(* Visualisation Lamp_status
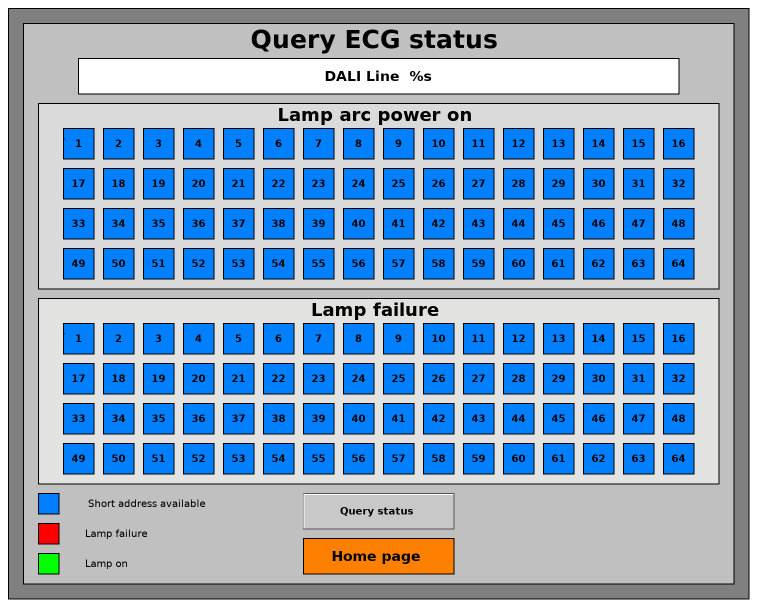
rectangle at (45,15)-(756,576): text "Query ECG status"
rounded rectangle at (325,530)-(476,566): text "Home page"; opens PLC_VISU; tooltip Back to home page
rounded rectangle at (100,50)-(701,86): text "DALI Line  %s"; shows DALI_Config.bDali_Linie; tooltip You can change the DALI Line only on the home page.
rectangle at (60,95)-(741,281): text "Lamp arc power on"
rectangle at (85,120)-(116,151): text "1"; alarm colour if DALI_Config.Kurzadr[1]
rectangle at (85,120)-(116,151): text "1"; invisible if not DALI_Config.Kurzadr[1]; alarm colour if DALI_Config.LampeEin[1]
rectangle at (125,120)-(156,151): text "2"; alarm colour if DALI_Config.Kurzadr[2]
rectangle at (125,120)-(156,151): text "2"; invisible if not DALI_Config.Kurzadr[2]; alarm colour if DALI_Config.LampeEin[2]
rectangle at (165,120)-(196,151): text "3"; alarm colour if DALI_Config.Kurzadr[3]
rectangle at (165,120)-(196,151): text "3"; invisible if not DALI_Config.Kurzadr[3]; alarm colour if DALI_Config.LampeEin[3]
rectangle at (205,120)-(236,151): text "4"; alarm colour if DALI_Config.Kurzadr[4]
rectangle at (205,120)-(236,151): text "4"; invisible if not DALI_Config.Kurzadr[4]; alarm colour if DALI_Config.LampeEin[4]
rectangle at (245,120)-(276,151): text "5"; alarm colour if DALI_Config.Kurzadr[5]
rectangle at (245,120)-(276,151): text "5"; invisible if not DALI_Config.Kurzadr[5]; alarm colour if DALI_Config.LampeEin[5]
rectangle at (285,120)-(316,151): text "6"; alarm colour if DALI_Config.Kurzadr[6]
rectangle at (285,120)-(316,151): text "6"; invisible if not DALI_Config.Kurzadr[6]; alarm colour if DALI_Config.LampeEin[6]
rectangle at (325,120)-(356,151): text "7"; alarm colour if DALI_Config.Kurzadr[7]
rectangle at (325,120)-(356,151): text "7"; invisible if not DALI_Config.Kurzadr[7]; alarm colour if DALI_Config.LampeEin[7]
rectangle at (365,120)-(396,151): text "8"; alarm colour if DALI_Config.Kurzadr[8]
rectangle at (365,120)-(396,151): text "8"; invisible if not DALI_Config.Kurzadr[8]; alarm colour if DALI_Config.LampeEin[8]
rectangle at (405,120)-(436,151): text "9"; alarm colour if DALI_Config.Kurzadr[9]
rectangle at (405,120)-(436,151): text "9"; invisible if not DALI_Config.Kurzadr[9]; alarm colour if DALI_Config.LampeEin[9]
rectangle at (445,120)-(476,151): text "10"; alarm colour if DALI_Config.Kurzadr[10]
rectangle at (445,120)-(476,151): text "10"; invisible if not DALI_Config.Kurzadr[10]; alarm colour if DALI_Config.LampeEin[10]
rectangle at (485,120)-(516,151): text "11"; alarm colour if DALI_Config.Kurzadr[11]
rectangle at (485,120)-(516,151): text "11"; invisible if not DALI_Config.Kurzadr[11]; alarm colour if DALI_Config.LampeEin[11]
rectangle at (525,120)-(556,151): text "12"; alarm colour if DALI_Config.Kurzadr[12]
rectangle at (525,120)-(556,151): text "12"; invisible if not DALI_Config.Kurzadr[12]; alarm colour if DALI_Config.LampeEin[12]
rectangle at (565,120)-(596,151): text "13"; alarm colour if DALI_Config.Kurzadr[13]
rectangle at (565,120)-(596,151): text "13"; invisible if not DALI_Config.Kurzadr[13]; alarm colour if DALI_Config.LampeEin[13]
rectangle at (605,120)-(636,151): text "14"; alarm colour if DALI_Config.Kurzadr[14]
rectangle at (605,120)-(636,151): text "14"; invisible if not DALI_Config.Kurzadr[14]; alarm colour if DALI_Config.LampeEin[14]
rectangle at (645,120)-(676,151): text "15"; alarm colour if DALI_Config.Kurzadr[15]
rectangle at (645,120)-(676,151): text "15"; invisible if not DALI_Config.Kurzadr[15]; alarm colour if DALI_Config.LampeEin[15]
rectangle at (685,120)-(716,151): text "16"; alarm colour if DALI_Config.Kurzadr[16]
rectangle at (685,120)-(716,151): text "16"; invisible if not DALI_Config.Kurzadr[16]; alarm colour if DALI_Config.LampeEin[16]
rectangle at (85,160)-(116,191): text "17"; alarm colour if DALI_Config.Kurzadr[17]
rectangle at (85,160)-(116,191): text "17"; invisible if not DALI_Config.Kurzadr[17]; alarm colour if DALI_Config.LampeEin[17]
rectangle at (165,160)-(196,191): text "19"; alarm colour if DALI_Config.Kurzadr[19]
rectangle at (165,160)-(196,191): text "19"; invisible if not DALI_Config.Kurzadr[19]; alarm colour if DALI_Config.LampeEin[19]
rectangle at (125,160)-(156,191): text "18"; alarm colour if DALI_Config.Kurzadr[18]
rectangle at (125,160)-(156,191): text "18"; invisible if not DALI_Config.Kurzadr[18]; alarm colour if DALI_Config.LampeEin[18]
rectangle at (205,160)-(236,191): text "20"; alarm colour if DALI_Config.Kurzadr[20]
rectangle at (205,160)-(236,191): text "20"; invisible if not DALI_Config.Kurzadr[20]; alarm colour if DALI_Config.LampeEin[20]
rectangle at (245,160)-(276,191): text "21"; alarm colour if DALI_Config.Kurzadr[21]
rectangle at (245,160)-(276,191): text "21"; invisible if not DALI_Config.Kurzadr[21]; alarm colour if DALI_Config.LampeEin[21]
rectangle at (285,160)-(316,191): text "22"; alarm colour if DALI_Config.Kurzadr[22]
rectangle at (285,160)-(316,191): text "22"; invisible if not DALI_Config.Kurzadr[22]; alarm colour if DALI_Config.LampeEin[22]
rectangle at (325,160)-(356,191): text "23"; alarm colour if DALI_Config.Kurzadr[23]
rectangle at (325,160)-(356,191): text "23"; invisible if not DALI_Config.Kurzadr[23]; alarm colour if DALI_Config.LampeEin[23]
rectangle at (365,160)-(396,191): text "24"; alarm colour if DALI_Config.Kurzadr[24]
rectangle at (365,160)-(396,191): text "24"; invisible if not DALI_Config.Kurzadr[24]; alarm colour if DALI_Config.LampeEin[24]
rectangle at (405,160)-(436,191): text "25"; alarm colour if DALI_Config.Kurzadr[25]
rectangle at (405,160)-(436,191): text "25"; invisible if not DALI_Config.Kurzadr[25]; alarm colour if DALI_Config.LampeEin[25]
rectangle at (565,160)-(596,191): text "29"; alarm colour if DALI_Config.Kurzadr[29]
rectangle at (565,160)-(596,191): text "29"; invisible if not DALI_Config.Kurzadr[29]; alarm colour if DALI_Config.LampeEin[29]
rectangle at (525,160)-(556,191): text "28"; alarm colour if DALI_Config.Kurzadr[28]
rectangle at (525,160)-(556,191): text "28"; invisible if not DALI_Config.Kurzadr[28]; alarm colour if DALI_Config.LampeEin[28]
rectangle at (485,160)-(516,191): text "27"; alarm colour if DALI_Config.Kurzadr[27]
rectangle at (485,160)-(516,191): text "27"; invisible if not DALI_Config.Kurzadr[27]; alarm colour if DALI_Config.LampeEin[27]
rectangle at (445,160)-(476,191): text "26"; alarm colour if DALI_Config.Kurzadr[26]
rectangle at (445,160)-(476,191): text "26"; invisible if not DALI_Config.Kurzadr[26]; alarm colour if DALI_Config.LampeEin[26]
rectangle at (605,160)-(636,191): text "30"; alarm colour if DALI_Config.Kurzadr[30]
rectangle at (605,160)-(636,191): text "30"; invisible if not DALI_Config.Kurzadr[30]; alarm colour if DALI_Config.LampeEin[30]
rectangle at (645,160)-(676,191): text "31"; alarm colour if DALI_Config.Kurzadr[31]
rectangle at (645,160)-(676,191): text "31"; invisible if not DALI_Config.Kurzadr[31]; alarm colour if DALI_Config.LampeEin[31]
rectangle at (685,160)-(716,191): text "32"; alarm colour if DALI_Config.Kurzadr[32]
rectangle at (685,160)-(716,191): text "32"; invisible if not DALI_Config.Kurzadr[32]; alarm colour if DALI_Config.LampeEin[32]
rectangle at (85,200)-(116,231): text "33"; alarm colour if DALI_Config.Kurzadr[33]
rectangle at (85,200)-(116,231): text "33"; invisible if not DALI_Config.Kurzadr[33]; alarm colour if DALI_Config.LampeEin[33]
rectangle at (125,200)-(156,231): text "34"; alarm colour if DALI_Config.Kurzadr[34]
rectangle at (125,200)-(156,231): text "34"; invisible if not DALI_Config.Kurzadr[34]; alarm colour if DALI_Config.LampeEin[34]
rectangle at (205,200)-(236,231): text "36"; alarm colour if DALI_Config.Kurzadr[36]
rectangle at (205,200)-(236,231): text "36"; invisible if not DALI_Config.Kurzadr[36]; alarm colour if DALI_Config.LampeEin[36]
rectangle at (285,200)-(316,231): text "38"; alarm colour if DALI_Config.Kurzadr[38]
rectangle at (285,200)-(316,231): text "38"; invisible if not DALI_Config.Kurzadr[38]; alarm colour if DALI_Config.LampeEin[38]
rectangle at (325,200)-(356,231): text "39"; alarm colour if DALI_Config.Kurzadr[39]
rectangle at (325,200)-(356,231): text "39"; invisible if not DALI_Config.Kurzadr[39]; alarm colour if DALI_Config.LampeEin[39]
rectangle at (245,200)-(276,231): text "37"; alarm colour if DALI_Config.Kurzadr[37]
rectangle at (245,200)-(276,231): text "37"; invisible if not DALI_Config.Kurzadr[37]; alarm colour if DALI_Config.LampeEin[37]
rectangle at (165,200)-(196,231): text "35"; alarm colour if DALI_Config.Kurzadr[35]
rectangle at (165,200)-(196,231): text "35"; invisible if not DALI_Config.Kurzadr[35]; alarm colour if DALI_Config.LampeEin[35]
rectangle at (405,200)-(436,231): text "41"; alarm colour if DALI_Config.Kurzadr[41]
rectangle at (405,200)-(436,231): text "41"; invisible if not DALI_Config.Kurzadr[41]; alarm colour if DALI_Config.LampeEin[41]
rectangle at (445,200)-(476,231): text "42"; alarm colour if DALI_Config.Kurzadr[42]
rectangle at (445,200)-(476,231): text "42"; invisible if not DALI_Config.Kurzadr[42]; alarm colour if DALI_Config.LampeEin[42]
rectangle at (365,200)-(396,231): text "40"; alarm colour if DALI_Config.Kurzadr[40]
rectangle at (365,200)-(396,231): text "40"; invisible if not DALI_Config.Kurzadr[40]; alarm colour if DALI_Config.LampeEin[40]
rectangle at (485,200)-(516,231): text "43"; alarm colour if DALI_Config.Kurzadr[43]
rectangle at (485,200)-(516,231): text "43"; invisible if not DALI_Config.Kurzadr[43]; alarm colour if DALI_Config.LampeEin[43]
rectangle at (525,200)-(556,231): text "44"; alarm colour if DALI_Config.Kurzadr[44]
rectangle at (525,200)-(556,231): text "44"; invisible if not DALI_Config.Kurzadr[44]; alarm colour if DALI_Config.LampeEin[44]
rectangle at (565,200)-(596,231): text "45"; alarm colour if DALI_Config.Kurzadr[45]
rectangle at (565,200)-(596,231): text "45"; invisible if not DALI_Config.Kurzadr[45]; alarm colour if DALI_Config.LampeEin[45]
rectangle at (605,200)-(636,231): text "46"; alarm colour if DALI_Config.Kurzadr[46]
rectangle at (605,200)-(636,231): text "46"; invisible if not DALI_Config.Kurzadr[46]; alarm colour if DALI_Config.LampeEin[46]
rectangle at (645,200)-(676,231): text "47"; alarm colour if DALI_Config.Kurzadr[47]
rectangle at (645,200)-(676,231): text "47"; invisible if not DALI_Config.Kurzadr[47]; alarm colour if DALI_Config.LampeEin[47]
rectangle at (685,200)-(716,231): text "48"; alarm colour if DALI_Config.Kurzadr[48]
rectangle at (685,200)-(716,231): text "48"; invisible if not DALI_Config.Kurzadr[48]; alarm colour if DALI_Config.LampeEin[48]
rectangle at (85,240)-(116,271): text "49"; alarm colour if DALI_Config.Kurzadr[49]
rectangle at (85,240)-(116,271): text "49"; invisible if not DALI_Config.Kurzadr[49]; alarm colour if DALI_Config.LampeEin[49]
rectangle at (125,240)-(156,271): text "50"; alarm colour if DALI_Config.Kurzadr[50]
rectangle at (125,240)-(156,271): text "50"; invisible if not DALI_Config.Kurzadr[50]; alarm colour if DALI_Config.LampeEin[50]
rectangle at (165,240)-(196,271): text "51"; alarm colour if DALI_Config.Kurzadr[51]
rectangle at (165,240)-(196,271): text "51"; invisible if not DALI_Config.Kurzadr[51]; alarm colour if DALI_Config.LampeEin[51]
rectangle at (205,240)-(236,271): text "52"; alarm colour if DALI_Config.Kurzadr[52]
rectangle at (205,240)-(236,271): text "52"; invisible if not DALI_Config.Kurzadr[52]; alarm colour if DALI_Config.LampeEin[52]
rectangle at (245,240)-(276,271): text "53"; alarm colour if DALI_Config.Kurzadr[53]
rectangle at (245,240)-(276,271): text "53"; invisible if not DALI_Config.Kurzadr[53]; alarm colour if DALI_Config.LampeEin[53]
rectangle at (285,240)-(316,271): text "54"; alarm colour if DALI_Config.Kurzadr[54]
rectangle at (285,240)-(316,271): text "54"; invisible if not DALI_Config.Kurzadr[54]; alarm colour if DALI_Config.LampeEin[54]
rectangle at (325,240)-(356,271): text "55"; alarm colour if DALI_Config.Kurzadr[55]
rectangle at (325,240)-(356,271): text "55"; invisible if not DALI_Config.Kurzadr[55]; alarm colour if DALI_Config.LampeEin[55]
rectangle at (365,240)-(396,271): text "56"; alarm colour if DALI_Config.Kurzadr[56]
rectangle at (365,240)-(396,271): text "56"; invisible if not DALI_Config.Kurzadr[56]; alarm colour if DALI_Config.LampeEin[56]
rectangle at (405,240)-(436,271): text "57"; alarm colour if DALI_Config.Kurzadr[57]
rectangle at (405,240)-(436,271): text "57"; invisible if not DALI_Config.Kurzadr[57]; alarm colour if DALI_Config.LampeEin[57]
rectangle at (485,240)-(516,271): text "59"; alarm colour if DALI_Config.Kurzadr[59]
rectangle at (485,240)-(516,271): text "59"; invisible if not DALI_Config.Kurzadr[59]; alarm colour if DALI_Config.LampeEin[59]
rectangle at (525,240)-(556,271): text "60"; alarm colour if DALI_Config.Kurzadr[60]
rectangle at (525,240)-(556,271): text "60"; invisible if not DALI_Config.Kurzadr[60]; alarm colour if DALI_Config.LampeEin[60]
rectangle at (565,240)-(596,271): text "61"; alarm colour if DALI_Config.Kurzadr[61]
rectangle at (565,240)-(596,271): text "61"; invisible if not DALI_Config.Kurzadr[61]; alarm colour if DALI_Config.LampeEin[61]
rectangle at (605,240)-(636,271): text "62"; alarm colour if DALI_Config.Kurzadr[62]
rectangle at (605,240)-(636,271): text "62"; invisible if not DALI_Config.Kurzadr[62]; alarm colour if DALI_Config.LampeEin[62]
rectangle at (445,240)-(476,271): text "58"; alarm colour if DALI_Config.Kurzadr[58]
rectangle at (445,240)-(476,271): text "58"; invisible if not DALI_Config.Kurzadr[58]; alarm colour if DALI_Config.LampeEin[58]
rectangle at (645,240)-(676,271): text "63"; alarm colour if DALI_Config.Kurzadr[63]
rectangle at (645,240)-(676,271): text "63"; invisible if not DALI_Config.Kurzadr[63]; alarm colour if DALI_Config.LampeEin[63]
rectangle at (685,240)-(716,271): text "64"; alarm colour if DALI_Config.Kurzadr[64]
rectangle at (685,240)-(716,271): text "64"; invisible if not DALI_Config.Kurzadr[64]; alarm colour if DALI_Config.LampeEin[64]
rectangle at (60,290)-(741,476): text "Lamp failure"
rectangle at (85,315)-(116,346): text "1"; alarm colour if DALI_Config.Kurzadr[1]
rectangle at (85,315)-(116,346): text "1"; invisible if not DALI_Config.Kurzadr[1]; alarm colour if DALI_Config.Lampenausfall[1]
rectangle at (125,315)-(156,346): text "2"; alarm colour if DALI_Config.Kurzadr[2]
rectangle at (125,315)-(156,346): text "2"; invisible if not DALI_Config.Kurzadr[2]; alarm colour if DALI_Config.Lampenausfall[2]
rectangle at (165,315)-(196,346): text "3"; alarm colour if DALI_Config.Kurzadr[3]
rectangle at (165,315)-(196,346): text "3"; invisible if not DALI_Config.Kurzadr[3]; alarm colour if DALI_Config.Lampenausfall[3]
rectangle at (205,315)-(236,346): text "4"; alarm colour if DALI_Config.Kurzadr[4]
rectangle at (205,315)-(236,346): text "4"; invisible if not DALI_Config.Kurzadr[4]; alarm colour if DALI_Config.Lampenausfall[4]
rectangle at (245,315)-(276,346): text "5"; alarm colour if DALI_Config.Kurzadr[5]
rectangle at (245,315)-(276,346): text "5"; invisible if not DALI_Config.Kurzadr[5]; alarm colour if DALI_Config.Lampenausfall[5]
rectangle at (285,315)-(316,346): text "6"; alarm colour if DALI_Config.Kurzadr[6]
rectangle at (285,315)-(316,346): text "6"; invisible if not DALI_Config.Kurzadr[6]; alarm colour if DALI_Config.Lampenausfall[6]
rectangle at (325,315)-(356,346): text "7"; alarm colour if DALI_Config.Kurzadr[7]
rectangle at (325,315)-(356,346): text "7"; invisible if not DALI_Config.Kurzadr[7]; alarm colour if DALI_Config.Lampenausfall[7]
rectangle at (365,315)-(396,346): text "8"; alarm colour if DALI_Config.Kurzadr[8]
rectangle at (365,315)-(396,346): text "8"; invisible if not DALI_Config.Kurzadr[8]; alarm colour if DALI_Config.Lampenausfall[8]
rectangle at (405,315)-(436,346): text "9"; alarm colour if DALI_Config.Kurzadr[9]
rectangle at (405,315)-(436,346): text "9"; invisible if not DALI_Config.Kurzadr[9]; alarm colour if DALI_Config.Lampenausfall[9]
rectangle at (445,315)-(476,346): text "10"; alarm colour if DALI_Config.Kurzadr[10]
rectangle at (445,315)-(476,346): text "10"; invisible if not DALI_Config.Kurzadr[10]; alarm colour if DALI_Config.Lampenausfall[10]
rectangle at (485,315)-(516,346): text "11"; alarm colour if DALI_Config.Kurzadr[11]
rectangle at (485,315)-(516,346): text "11"; invisible if not DALI_Config.Kurzadr[11]; alarm colour if DALI_Config.Lampenausfall[11]
rectangle at (525,315)-(556,346): text "12"; alarm colour if DALI_Config.Kurzadr[12]
rectangle at (525,315)-(556,346): text "12"; invisible if not DALI_Config.Kurzadr[12]; alarm colour if DALI_Config.Lampenausfall[12]
rectangle at (565,315)-(596,346): text "13"; alarm colour if DALI_Config.Kurzadr[13]
rectangle at (565,315)-(596,346): text "13"; invisible if not DALI_Config.Kurzadr[13]; alarm colour if DALI_Config.Lampenausfall[13]
rectangle at (605,315)-(636,346): text "14"; alarm colour if DALI_Config.Kurzadr[14]
rectangle at (605,315)-(636,346): text "14"; invisible if not DALI_Config.Kurzadr[14]; alarm colour if DALI_Config.Lampenausfall[14]
rectangle at (645,315)-(676,346): text "15"; alarm colour if DALI_Config.Kurzadr[15]
rectangle at (645,315)-(676,346): text "15"; invisible if not DALI_Config.Kurzadr[15]; alarm colour if DALI_Config.Lampenausfall[15]
rectangle at (685,315)-(716,346): text "16"; alarm colour if DALI_Config.Kurzadr[16]
rectangle at (685,315)-(716,346): text "16"; invisible if not DALI_Config.Kurzadr[16]; alarm colour if DALI_Config.Lampenausfall[16]
rectangle at (85,355)-(116,386): text "17"; alarm colour if DALI_Config.Kurzadr[17]
rectangle at (85,355)-(116,386): text "17"; invisible if not DALI_Config.Kurzadr[17]; alarm colour if DALI_Config.Lampenausfall[17]
rectangle at (165,355)-(196,386): text "19"; alarm colour if DALI_Config.Kurzadr[19]
rectangle at (165,355)-(196,386): text "19"; invisible if not DALI_Config.Kurzadr[19]; alarm colour if DALI_Config.Lampenausfall[19]
rectangle at (125,355)-(156,386): text "18"; alarm colour if DALI_Config.Kurzadr[18]
rectangle at (125,355)-(156,386): text "18"; invisible if not DALI_Config.Kurzadr[18]; alarm colour if DALI_Config.Lampenausfall[18]
rectangle at (205,355)-(236,386): text "20"; alarm colour if DALI_Config.Kurzadr[20]
rectangle at (205,355)-(236,386): text "20"; invisible if not DALI_Config.Kurzadr[20]; alarm colour if DALI_Config.Lampenausfall[20]
rectangle at (245,355)-(276,386): text "21"; alarm colour if DALI_Config.Kurzadr[21]
rectangle at (245,355)-(276,386): text "21"; invisible if not DALI_Config.Kurzadr[21]; alarm colour if DALI_Config.Lampenausfall[21]
rectangle at (285,355)-(316,386): text "22"; alarm colour if DALI_Config.Kurzadr[22]
rectangle at (285,355)-(316,386): text "22"; invisible if not DALI_Config.Kurzadr[22]; alarm colour if DALI_Config.Lampenausfall[22]
rectangle at (325,355)-(356,386): text "23"; alarm colour if DALI_Config.Kurzadr[23]
rectangle at (325,355)-(356,386): text "23"; invisible if not DALI_Config.Kurzadr[23]; alarm colour if DALI_Config.Lampenausfall[23]
rectangle at (365,355)-(396,386): text "24"; alarm colour if DALI_Config.Kurzadr[24]
rectangle at (365,355)-(396,386): text "24"; invisible if not DALI_Config.Kurzadr[24]; alarm colour if DALI_Config.Lampenausfall[24]
rectangle at (405,355)-(436,386): text "25"; alarm colour if DALI_Config.Kurzadr[25]
rectangle at (405,355)-(436,386): text "25"; invisible if not DALI_Config.Kurzadr[25]; alarm colour if DALI_Config.Lampenausfall[25]
rectangle at (565,355)-(596,386): text "29"; alarm colour if DALI_Config.Kurzadr[29]
rectangle at (565,355)-(596,386): text "29"; invisible if not DALI_Config.Kurzadr[29]; alarm colour if DALI_Config.Lampenausfall[29]
rectangle at (525,355)-(556,386): text "28"; alarm colour if DALI_Config.Kurzadr[28]
rectangle at (525,355)-(556,386): text "28"; invisible if not DALI_Config.Kurzadr[28]; alarm colour if DALI_Config.Lampenausfall[28]
rectangle at (485,355)-(516,386): text "27"; alarm colour if DALI_Config.Kurzadr[27]
rectangle at (485,355)-(516,386): text "27"; invisible if not DALI_Config.Kurzadr[27]; alarm colour if DALI_Config.Lampenausfall[27]
rectangle at (445,355)-(476,386): text "26"; alarm colour if DALI_Config.Kurzadr[26]
rectangle at (445,355)-(476,386): text "26"; invisible if not DALI_Config.Kurzadr[26]; alarm colour if DALI_Config.Lampenausfall[26]
rectangle at (605,355)-(636,386): text "30"; alarm colour if DALI_Config.Kurzadr[30]
rectangle at (605,355)-(636,386): text "30"; invisible if not DALI_Config.Kurzadr[30]; alarm colour if DALI_Config.Lampenausfall[30]
rectangle at (645,355)-(676,386): text "31"; alarm colour if DALI_Config.Kurzadr[31]
rectangle at (645,355)-(676,386): text "31"; invisible if not DALI_Config.Kurzadr[31]; alarm colour if DALI_Config.Lampenausfall[31]
rectangle at (685,355)-(716,386): text "32"; alarm colour if DALI_Config.Kurzadr[32]
rectangle at (685,355)-(716,386): text "32"; invisible if not DALI_Config.Kurzadr[32]; alarm colour if DALI_Config.Lampenausfall[32]
rectangle at (85,395)-(116,426): text "33"; alarm colour if DALI_Config.Kurzadr[33]
rectangle at (85,395)-(116,426): text "33"; invisible if not DALI_Config.Kurzadr[33]; alarm colour if DALI_Config.Lampenausfall[33]
rectangle at (125,395)-(156,426): text "34"; alarm colour if DALI_Config.Kurzadr[34]
rectangle at (125,395)-(156,426): text "34"; invisible if not DALI_Config.Kurzadr[34]; alarm colour if DALI_Config.Lampenausfall[34]
rectangle at (205,395)-(236,426): text "36"; alarm colour if DALI_Config.Kurzadr[36]
rectangle at (205,395)-(236,426): text "36"; invisible if not DALI_Config.Kurzadr[36]; alarm colour if DALI_Config.Lampenausfall[36]
rectangle at (285,395)-(316,426): text "38"; alarm colour if DALI_Config.Kurzadr[38]
rectangle at (285,395)-(316,426): text "38"; invisible if not DALI_Config.Kurzadr[38]; alarm colour if DALI_Config.Lampenausfall[38]
rectangle at (325,395)-(356,426): text "39"; alarm colour if DALI_Config.Kurzadr[39]
rectangle at (325,395)-(356,426): text "39"; invisible if not DALI_Config.Kurzadr[39]; alarm colour if DALI_Config.Lampenausfall[39]
rectangle at (245,395)-(276,426): text "37"; alarm colour if DALI_Config.Kurzadr[37]
rectangle at (245,395)-(276,426): text "37"; invisible if not DALI_Config.Kurzadr[37]; alarm colour if DALI_Config.Lampenausfall[37]
rectangle at (165,395)-(196,426): text "35"; alarm colour if DALI_Config.Kurzadr[35]
rectangle at (165,395)-(196,426): text "35"; invisible if not DALI_Config.Kurzadr[35]; alarm colour if DALI_Config.Lampenausfall[35]
rectangle at (405,395)-(436,426): text "41"; alarm colour if DALI_Config.Kurzadr[41]
rectangle at (405,395)-(436,426): text "41"; invisible if not DALI_Config.Kurzadr[41]; alarm colour if DALI_Config.Lampenausfall[41]
rectangle at (445,395)-(476,426): text "42"; alarm colour if DALI_Config.Kurzadr[42]
rectangle at (445,395)-(476,426): text "42"; invisible if not DALI_Config.Kurzadr[42]; alarm colour if DALI_Config.Lampenausfall[42]
rectangle at (365,395)-(396,426): text "40"; alarm colour if DALI_Config.Kurzadr[40]
rectangle at (365,395)-(396,426): text "40"; invisible if not DALI_Config.Kurzadr[40]; alarm colour if DALI_Config.Lampenausfall[40]
rectangle at (485,395)-(516,426): text "43"; alarm colour if DALI_Config.Kurzadr[43]
rectangle at (485,395)-(516,426): text "43"; invisible if not DALI_Config.Kurzadr[43]; alarm colour if DALI_Config.Lampenausfall[43]
rectangle at (525,395)-(556,426): text "44"; alarm colour if DALI_Config.Kurzadr[44]
rectangle at (525,395)-(556,426): text "44"; invisible if not DALI_Config.Kurzadr[44]; alarm colour if DALI_Config.Lampenausfall[44]
rectangle at (565,395)-(596,426): text "45"; alarm colour if DALI_Config.Kurzadr[45]
rectangle at (565,395)-(596,426): text "45"; invisible if not DALI_Config.Kurzadr[45]; alarm colour if DALI_Config.Lampenausfall[45]
rectangle at (605,395)-(636,426): text "46"; alarm colour if DALI_Config.Kurzadr[46]
rectangle at (605,395)-(636,426): text "46"; invisible if not DALI_Config.Kurzadr[46]; alarm colour if DALI_Config.Lampenausfall[46]
rectangle at (645,395)-(676,426): text "47"; alarm colour if DALI_Config.Kurzadr[47]
rectangle at (645,395)-(676,426): text "47"; invisible if not DALI_Config.Kurzadr[47]; alarm colour if DALI_Config.Lampenausfall[47]
rectangle at (685,395)-(716,426): text "48"; alarm colour if DALI_Config.Kurzadr[48]
rectangle at (685,395)-(716,426): text "48"; invisible if not DALI_Config.Kurzadr[48]; alarm colour if DALI_Config.Lampenausfall[48]
rectangle at (85,435)-(116,466): text "49"; alarm colour if DALI_Config.Kurzadr[49]
rectangle at (85,435)-(116,466): text "49"; invisible if not DALI_Config.Kurzadr[49]; alarm colour if DALI_Config.Lampenausfall[49]
rectangle at (125,435)-(156,466): text "50"; alarm colour if DALI_Config.Kurzadr[50]
rectangle at (125,435)-(156,466): text "50"; invisible if not DALI_Config.Kurzadr[50]; alarm colour if DALI_Config.Lampenausfall[50]
rectangle at (165,435)-(196,466): text "51"; alarm colour if DALI_Config.Kurzadr[51]
rectangle at (165,435)-(196,466): text "51"; invisible if not DALI_Config.Kurzadr[51]; alarm colour if DALI_Config.Lampenausfall[51]
rectangle at (205,435)-(236,466): text "52"; alarm colour if DALI_Config.Kurzadr[52]
rectangle at (205,435)-(236,466): text "52"; invisible if not DALI_Config.Kurzadr[52]; alarm colour if DALI_Config.Lampenausfall[52]
rectangle at (245,435)-(276,466): text "53"; alarm colour if DALI_Config.Kurzadr[53]
rectangle at (245,435)-(276,466): text "53"; invisible if not DALI_Config.Kurzadr[53]; alarm colour if DALI_Config.Lampenausfall[53]
rectangle at (285,435)-(316,466): text "54"; alarm colour if DALI_Config.Kurzadr[54]
rectangle at (285,435)-(316,466): text "54"; invisible if not DALI_Config.Kurzadr[54]; alarm colour if DALI_Config.Lampenausfall[54]
rectangle at (325,435)-(356,466): text "55"; alarm colour if DALI_Config.Kurzadr[55]
rectangle at (325,435)-(356,466): text "55"; invisible if not DALI_Config.Kurzadr[55]; alarm colour if DALI_Config.Lampenausfall[55]
rectangle at (365,435)-(396,466): text "56"; alarm colour if DALI_Config.Kurzadr[56]
rectangle at (365,435)-(396,466): text "56"; invisible if not DALI_Config.Kurzadr[56]; alarm colour if DALI_Config.Lampenausfall[56]
rectangle at (405,435)-(436,466): text "57"; alarm colour if DALI_Config.Kurzadr[57]
rectangle at (405,435)-(436,466): text "57"; invisible if not DALI_Config.Kurzadr[57]; alarm colour if DALI_Config.Lampenausfall[57]
rectangle at (485,435)-(516,466): text "59"; alarm colour if DALI_Config.Kurzadr[59]
rectangle at (485,435)-(516,466): text "59"; invisible if not DALI_Config.Kurzadr[59]; alarm colour if DALI_Config.Lampenausfall[59]
rectangle at (525,435)-(556,466): text "60"; alarm colour if DALI_Config.Kurzadr[60]
rectangle at (525,435)-(556,466): text "60"; invisible if not DALI_Config.Kurzadr[60]; alarm colour if DALI_Config.Lampenausfall[60]
rectangle at (565,435)-(596,466): text "61"; alarm colour if DALI_Config.Kurzadr[61]
rectangle at (565,435)-(596,466): text "61"; invisible if not DALI_Config.Kurzadr[61]; alarm colour if DALI_Config.Lampenausfall[61]
rectangle at (605,435)-(636,466): text "62"; alarm colour if DALI_Config.Kurzadr[62]
rectangle at (605,435)-(636,466): text "62"; invisible if not DALI_Config.Kurzadr[62]; alarm colour if DALI_Config.Lampenausfall[62]
rectangle at (445,435)-(476,466): text "58"; alarm colour if DALI_Config.Kurzadr[58]
rectangle at (445,435)-(476,466): text "58"; invisible if not DALI_Config.Kurzadr[58]; alarm colour if DALI_Config.Lampenausfall[58]
rectangle at (645,435)-(676,466): text "63"; alarm colour if DALI_Config.Kurzadr[63]
rectangle at (645,435)-(676,466): text "63"; invisible if not DALI_Config.Kurzadr[63]; alarm colour if DALI_Config.Lampenausfall[63]
rectangle at (685,435)-(716,466): text "64"; alarm colour if DALI_Config.Kurzadr[64]
rectangle at (685,435)-(716,466): text "64"; invisible if not DALI_Config.Kurzadr[64]; alarm colour if DALI_Config.Lampenausfall[64]
button at (325,485)-(476,521): text "Query status"; taps DALI_Config.Status; tooltip If you click the button "Query Status", you will get the status "Lamp failure" and "Lamp arc power on" from the ECG.
rectangle at (90,485)-(251,506): text "Short address available"
rectangle at (105,515)-(236,536): text "Lamp failure"
rectangle at (105,545)-(176,566): text "Lamp on"
6 more shapes without text or variables
*)

(* Visualisation PLC_VISU
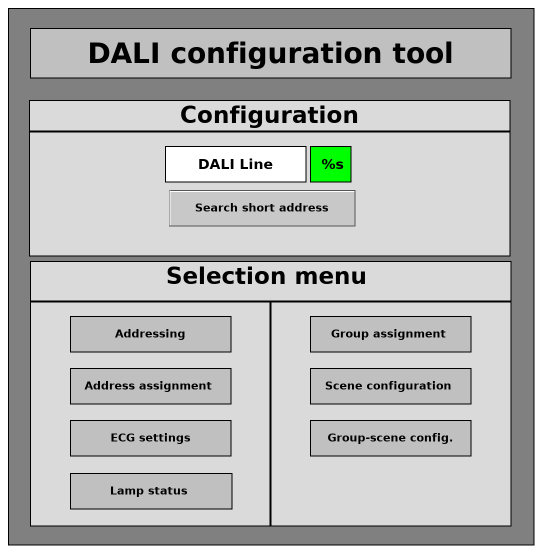
rectangle at (170,100)-(651,256): text "Configuration"
rectangle at (171,261)-(652,526): text "Selection menu"
rectangle at (171,28)-(652,78): text "DALI configuration tool"
rectangle at (211,316)-(372,352): text "Addressing"; opens Addressing
rectangle at (211,368)-(372,404): text "Address assignment"; opens Sort_short_address
rectangle at (451,316)-(612,352): text "Group assignment"; opens group_assignment
rectangle at (451,368)-(612,404): text "Scene configuration"; opens Scene_configuration
rectangle at (211,420)-(372,456): text "ECG settings"; opens ECG_settings
rectangle at (451,420)-(612,456): text "Group-scene config."; opens GroupSceneConfiguration
rectangle at (306,146)-(447,182): text "DALI Line"
button at (310,190)-(496,226): text "Search short address"; taps DALI_Config.SucheKurzadr; tooltip Clicking the button "Search Short Address" will start the search for available short addresses.
rectangle at (451,146)-(492,182): text "%s"; shows DALI_Config.Dali_Linie; alarm colour if DALI_Config.keineJobliste; tooltip Select DALI Line (1 - 5); editable
rectangle at (211,473)-(373,509): text "Lamp status"; opens Lamp_status
4 more shapes without text or variables
*)

(* Visualisation Scene_configuration
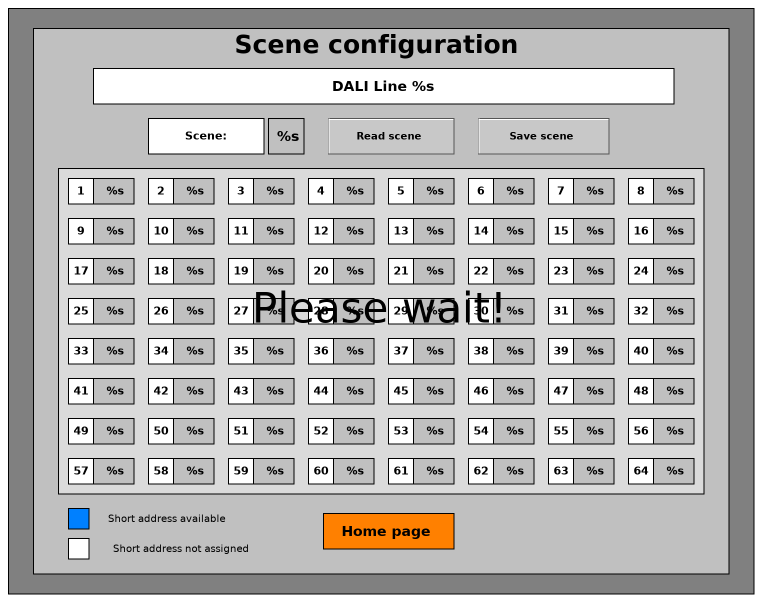
rectangle at (50,25)-(746,571): text "Scene configuration"
rounded rectangle at (340,510)-(471,546): text "Home page"; opens PLC_VISU; tooltip Back to home page
rounded rectangle at (110,65)-(691,101): text "DALI Line %s"; shows DALI_Config.bDali_Linie; tooltip You can change the DALI Line only on the home page.
rectangle at (85,175)-(111,201): text "1"; alarm colour if Dali_Config.Kurzadr[1]
rectangle at (110,175)-(151,201): text "%s"; shows DALI_Config.Szenenwert[1]; tooltip 0 % = Off 1 - 100 % = Dim level 101 % = Mask; editable
button at (495,115)-(626,151): text "Save scene"; taps DALI_Config.SzeneSpeichern; tooltip Save the configured dim levels in the ECGs.
button at (345,115)-(471,151): text "Read scene"; taps DALI_Config.SzeneLesen; tooltip Read the saved scene values from the ECGs.
rectangle at (85,215)-(111,241): text "9"; alarm colour if Dali_Config.Kurzadr[9]
rectangle at (110,215)-(151,241): text "%s"; shows DALI_Config.Szenenwert[9]; tooltip 0 % = Off 1 - 100 % = Dim level 101 % = Mask; editable
rectangle at (85,255)-(111,281): text "17"; alarm colour if Dali_Config.Kurzadr[17]
rectangle at (110,255)-(151,281): text "%s"; shows DALI_Config.Szenenwert[17]; tooltip 0 % = Off 1 - 100 % = Dim level 101 % = Mask; editable
rectangle at (85,295)-(111,321): text "25"; alarm colour if Dali_Config.Kurzadr[25]
rectangle at (110,295)-(151,321): text "%s"; shows DALI_Config.Szenenwert[25]; tooltip 0 % = Off 1 - 100 % = Dim level 101 % = Mask; editable
rectangle at (85,335)-(111,361): text "33"; alarm colour if Dali_Config.Kurzadr[33]
rectangle at (110,335)-(151,361): text "%s"; shows DALI_Config.Szenenwert[33]; tooltip 0 % = Off 1 - 100 % = Dim level 101 % = Mask; editable
rectangle at (85,375)-(111,401): text "41"; alarm colour if Dali_Config.Kurzadr[41]
rectangle at (110,375)-(151,401): text "%s"; shows DALI_Config.Szenenwert[41]; tooltip 0 % = Off 1 - 100 % = Dim level 101 % = Mask; editable
rectangle at (85,415)-(111,441): text "49"; alarm colour if Dali_Config.Kurzadr[49]
rectangle at (110,415)-(151,441): text "%s"; shows DALI_Config.Szenenwert[49]; tooltip 0 % = Off 1 - 100 % = Dim level 101 % = Mask; editable
rectangle at (85,455)-(111,481): text "57"; alarm colour if Dali_Config.Kurzadr[57]
rectangle at (110,455)-(151,481): text "%s"; shows DALI_Config.Szenenwert[57]; tooltip 0 % = Off 1 - 100 % = Dim level 101 % = Mask; editable
rectangle at (165,175)-(191,201): text "2"; alarm colour if Dali_Config.Kurzadr[2]
rectangle at (190,175)-(231,201): text "%s"; shows DALI_Config.Szenenwert[2]; tooltip 0 % = Off 1 - 100 % = Dim level 101 % = Mask; editable
rectangle at (165,215)-(191,241): text "10"; alarm colour if Dali_Config.Kurzadr[10]
rectangle at (190,215)-(231,241): text "%s"; shows DALI_Config.Szenenwert[10]; tooltip 0 % = Off 1 - 100 % = Dim level 101 % = Mask; editable
rectangle at (165,255)-(191,281): text "18"; alarm colour if Dali_Config.Kurzadr[18]
rectangle at (190,255)-(231,281): text "%s"; shows DALI_Config.Szenenwert[18]; tooltip 0 % = Off 1 - 100 % = Dim level 101 % = Mask; editable
rectangle at (165,295)-(191,321): text "26"; alarm colour if Dali_Config.Kurzadr[26]
rectangle at (190,295)-(231,321): text "%s"; shows DALI_Config.Szenenwert[26]; tooltip 0 % = Off 1 - 100 % = Dim level 101 % = Mask; editable
rectangle at (165,335)-(191,361): text "34"; alarm colour if Dali_Config.Kurzadr[34]
rectangle at (190,335)-(231,361): text "%s"; shows DALI_Config.Szenenwert[34]; tooltip 0 % = Off 1 - 100 % = Dim level 101 % = Mask; editable
rectangle at (165,375)-(191,401): text "42"; alarm colour if Dali_Config.Kurzadr[42]
rectangle at (190,375)-(231,401): text "%s"; shows DALI_Config.Szenenwert[42]; tooltip 0 % = Off 1 - 100 % = Dim level 101 % = Mask; editable
rectangle at (165,415)-(191,441): text "50"; alarm colour if Dali_Config.Kurzadr[50]
rectangle at (190,415)-(231,441): text "%s"; shows DALI_Config.Szenenwert[50]; tooltip 0 % = Off 1 - 100 % = Dim level 101 % = Mask; editable
rectangle at (165,455)-(191,481): text "58"; alarm colour if Dali_Config.Kurzadr[58]
rectangle at (190,455)-(231,481): text "%s"; shows DALI_Config.Szenenwert[58]; tooltip 0 % = Off 1 - 100 % = Dim level 101 % = Mask; editable
rectangle at (245,175)-(271,201): text "3"; alarm colour if Dali_Config.Kurzadr[3]
rectangle at (270,175)-(311,201): text "%s"; shows DALI_Config.Szenenwert[3]; tooltip 0 % = Off 1 - 100 % = Dim level 101 % = Mask; editable
rectangle at (245,215)-(271,241): text "11"; alarm colour if Dali_Config.Kurzadr[11]
rectangle at (270,215)-(311,241): text "%s"; shows DALI_Config.Szenenwert[11]; tooltip 0 % = Off 1 - 100 % = Dim level 101 % = Mask; editable
rectangle at (245,255)-(271,281): text "19"; alarm colour if Dali_Config.Kurzadr[19]
rectangle at (270,255)-(311,281): text "%s"; shows DALI_Config.Szenenwert[19]; tooltip 0 % = Off 1 - 100 % = Dim level 101 % = Mask; editable
rectangle at (245,295)-(271,321): text "27"; alarm colour if Dali_Config.Kurzadr[27]
rectangle at (270,295)-(311,321): text "%s"; shows DALI_Config.Szenenwert[27]; tooltip 0 % = Off 1 - 100 % = Dim level 101 % = Mask; editable
rectangle at (245,335)-(271,361): text "35"; alarm colour if Dali_Config.Kurzadr[35]
rectangle at (270,335)-(311,361): text "%s"; shows DALI_Config.Szenenwert[35]; tooltip 0 % = Off 1 - 100 % = Dim level 101 % = Mask; editable
rectangle at (245,375)-(271,401): text "43"; alarm colour if Dali_Config.Kurzadr[43]
rectangle at (270,375)-(311,401): text "%s"; shows DALI_Config.Szenenwert[43]; tooltip 0 % = Off 1 - 100 % = Dim level 101 % = Mask; editable
rectangle at (245,415)-(271,441): text "51"; alarm colour if Dali_Config.Kurzadr[51]
rectangle at (270,415)-(311,441): text "%s"; shows DALI_Config.Szenenwert[51]; tooltip 0 % = Off 1 - 100 % = Dim level 101 % = Mask; editable
rectangle at (245,455)-(271,481): text "59"; alarm colour if Dali_Config.Kurzadr[59]
rectangle at (270,455)-(311,481): text "%s"; shows DALI_Config.Szenenwert[59]; tooltip 0 % = Off 1 - 100 % = Dim level 101 % = Mask; editable
rectangle at (325,175)-(351,201): text "4"; alarm colour if Dali_Config.Kurzadr[4]
rectangle at (350,175)-(391,201): text "%s"; shows DALI_Config.Szenenwert[4]; tooltip 0 % = Off 1 - 100 % = Dim level 101 % = Mask; editable
rectangle at (325,215)-(351,241): text "12"; alarm colour if Dali_Config.Kurzadr[12]
rectangle at (350,215)-(391,241): text "%s"; shows DALI_Config.Szenenwert[12]; tooltip 0 % = Off 1 - 100 % = Dim level 101 % = Mask; editable
rectangle at (325,255)-(351,281): text "20"; alarm colour if Dali_Config.Kurzadr[20]
rectangle at (350,255)-(391,281): text "%s"; shows DALI_Config.Szenenwert[20]; tooltip 0 % = Off 1 - 100 % = Dim level 101 % = Mask; editable
rectangle at (325,295)-(351,321): text "28"; alarm colour if Dali_Config.Kurzadr[28]
rectangle at (350,295)-(391,321): text "%s"; shows DALI_Config.Szenenwert[28]; tooltip 0 % = Off 1 - 100 % = Dim level 101 % = Mask; editable
rectangle at (325,335)-(351,361): text "36"; alarm colour if Dali_Config.Kurzadr[36]
rectangle at (350,335)-(391,361): text "%s"; shows DALI_Config.Szenenwert[36]; tooltip 0 % = Off 1 - 100 % = Dim level 101 % = Mask; editable
rectangle at (325,375)-(351,401): text "44"; alarm colour if Dali_Config.Kurzadr[44]
rectangle at (350,375)-(391,401): text "%s"; shows DALI_Config.Szenenwert[44]; tooltip 0 % = Off 1 - 100 % = Dim level 101 % = Mask; editable
rectangle at (325,415)-(351,441): text "52"; alarm colour if Dali_Config.Kurzadr[52]
rectangle at (350,415)-(391,441): text "%s"; shows DALI_Config.Szenenwert[52]; tooltip 0 % = Off 1 - 100 % = Dim level 101 % = Mask; editable
rectangle at (325,455)-(351,481): text "60"; alarm colour if Dali_Config.Kurzadr[60]
rectangle at (350,455)-(391,481): text "%s"; shows DALI_Config.Szenenwert[60]; tooltip 0 % = Off 1 - 100 % = Dim level 101 % = Mask; editable
rectangle at (405,175)-(431,201): text "5"; alarm colour if Dali_Config.Kurzadr[5]
rectangle at (430,175)-(471,201): text "%s"; shows DALI_Config.Szenenwert[5]; tooltip 0 % = Off 1 - 100 % = Dim level 101 % = Mask; editable
rectangle at (405,215)-(431,241): text "13"; alarm colour if Dali_Config.Kurzadr[13]
rectangle at (430,215)-(471,241): text "%s"; shows DALI_Config.Szenenwert[13]; tooltip 0 % = Off 1 - 100 % = Dim level 101 % = Mask; editable
rectangle at (405,255)-(431,281): text "21"; alarm colour if Dali_Config.Kurzadr[21]
rectangle at (430,255)-(471,281): text "%s"; shows DALI_Config.Szenenwert[21]; tooltip 0 % = Off 1 - 100 % = Dim level 101 % = Mask; editable
rectangle at (405,295)-(431,321): text "29"; alarm colour if Dali_Config.Kurzadr[29]
rectangle at (430,295)-(471,321): text "%s"; shows DALI_Config.Szenenwert[29]; tooltip 0 % = Off 1 - 100 % = Dim level 101 % = Mask; editable
rectangle at (405,335)-(431,361): text "37"; alarm colour if Dali_Config.Kurzadr[37]
rectangle at (430,335)-(471,361): text "%s"; shows DALI_Config.Szenenwert[37]; tooltip 0 % = Off 1 - 100 % = Dim level 101 % = Mask; editable
rectangle at (405,375)-(431,401): text "45"; alarm colour if Dali_Config.Kurzadr[45]
rectangle at (430,375)-(471,401): text "%s"; shows DALI_Config.Szenenwert[45]; tooltip 0 % = Off 1 - 100 % = Dim level 101 % = Mask; editable
rectangle at (405,415)-(431,441): text "53"; alarm colour if Dali_Config.Kurzadr[53]
rectangle at (430,415)-(471,441): text "%s"; shows DALI_Config.Szenenwert[53]; tooltip 0 % = Off 1 - 100 % = Dim level 101 % = Mask; editable
rectangle at (405,455)-(431,481): text "61"; alarm colour if Dali_Config.Kurzadr[61]
rectangle at (430,455)-(471,481): text "%s"; shows DALI_Config.Szenenwert[61]; tooltip 0 % = Off 1 - 100 % = Dim level 101 % = Mask; editable
rectangle at (485,175)-(511,201): text "6"; alarm colour if Dali_Config.Kurzadr[6]
rectangle at (510,175)-(551,201): text "%s"; shows DALI_Config.Szenenwert[6]; tooltip 0 % = Off 1 - 100 % = Dim level 101 % = Mask; editable
rectangle at (485,215)-(511,241): text "14"; alarm colour if Dali_Config.Kurzadr[14]
rectangle at (510,215)-(551,241): text "%s"; shows DALI_Config.Szenenwert[14]; tooltip 0 % = Off 1 - 100 % = Dim level 101 % = Mask; editable
rectangle at (485,255)-(511,281): text "22"; alarm colour if Dali_Config.Kurzadr[22]
rectangle at (510,255)-(551,281): text "%s"; shows DALI_Config.Szenenwert[22]; tooltip 0 % = Off 1 - 100 % = Dim level 101 % = Mask; editable
rectangle at (485,295)-(511,321): text "30"; alarm colour if Dali_Config.Kurzadr[30]
rectangle at (510,295)-(551,321): text "%s"; shows DALI_Config.Szenenwert[30]; tooltip 0 % = Off 1 - 100 % = Dim level 101 % = Mask; editable
rectangle at (485,335)-(511,361): text "38"; alarm colour if Dali_Config.Kurzadr[38]
rectangle at (510,335)-(551,361): text "%s"; shows DALI_Config.Szenenwert[38]; tooltip 0 % = Off 1 - 100 % = Dim level 101 % = Mask; editable
rectangle at (485,375)-(511,401): text "46"; alarm colour if Dali_Config.Kurzadr[46]
rectangle at (510,375)-(551,401): text "%s"; shows DALI_Config.Szenenwert[46]; tooltip 0 % = Off 1 - 100 % = Dim level 101 % = Mask; editable
rectangle at (485,415)-(511,441): text "54"; alarm colour if Dali_Config.Kurzadr[54]
rectangle at (510,415)-(551,441): text "%s"; shows DALI_Config.Szenenwert[54]; tooltip 0 % = Off 1 - 100 % = Dim level 101 % = Mask; editable
rectangle at (485,455)-(511,481): text "62"; alarm colour if Dali_Config.Kurzadr[62]
rectangle at (510,455)-(551,481): text "%s"; shows DALI_Config.Szenenwert[62]; tooltip 0 % = Off 1 - 100 % = Dim level 101 % = Mask; editable
rectangle at (565,175)-(591,201): text "7"; alarm colour if Dali_Config.Kurzadr[7]
rectangle at (590,175)-(631,201): text "%s"; shows DALI_Config.Szenenwert[7]; tooltip 0 % = Off 1 - 100 % = Dim level 101 % = Mask; editable
rectangle at (565,215)-(591,241): text "15"; alarm colour if Dali_Config.Kurzadr[15]
rectangle at (590,215)-(631,241): text "%s"; shows DALI_Config.Szenenwert[15]; tooltip 0 % = Off 1 - 100 % = Dim level 101 % = Mask; editable
rectangle at (565,255)-(591,281): text "23"; alarm colour if Dali_Config.Kurzadr[23]
rectangle at (590,255)-(631,281): text "%s"; shows DALI_Config.Szenenwert[23]; tooltip 0 % = Off 1 - 100 % = Dim level 101 % = Mask; editable
rectangle at (565,295)-(591,321): text "31"; alarm colour if Dali_Config.Kurzadr[31]
rectangle at (590,295)-(631,321): text "%s"; shows DALI_Config.Szenenwert[31]; tooltip 0 % = Off 1 - 100 % = Dim level 101 % = Mask; editable
rectangle at (565,335)-(591,361): text "39"; alarm colour if Dali_Config.Kurzadr[39]
rectangle at (590,335)-(631,361): text "%s"; shows DALI_Config.Szenenwert[39]; tooltip 0 % = Off 1 - 100 % = Dim level 101 % = Mask; editable
rectangle at (565,375)-(591,401): text "47"; alarm colour if Dali_Config.Kurzadr[47]
rectangle at (590,375)-(631,401): text "%s"; shows DALI_Config.Szenenwert[47]; tooltip 0 % = Off 1 - 100 % = Dim level 101 % = Mask; editable
rectangle at (565,415)-(591,441): text "55"; alarm colour if Dali_Config.Kurzadr[55]
rectangle at (590,415)-(631,441): text "%s"; shows DALI_Config.Szenenwert[55]; tooltip 0 % = Off 1 - 100 % = Dim level 101 % = Mask; editable
rectangle at (565,455)-(591,481): text "63"; alarm colour if Dali_Config.Kurzadr[63]
rectangle at (590,455)-(631,481): text "%s"; shows DALI_Config.Szenenwert[63]; tooltip 0 % = Off 1 - 100 % = Dim level 101 % = Mask; editable
rectangle at (645,175)-(671,201): text "8"; alarm colour if Dali_Config.Kurzadr[8]
rectangle at (670,175)-(711,201): text "%s"; shows DALI_Config.Szenenwert[8]; tooltip 0 % = Off 1 - 100 % = Dim level 101 % = Mask; editable
rectangle at (645,215)-(671,241): text "16"; alarm colour if Dali_Config.Kurzadr[16]
rectangle at (670,215)-(711,241): text "%s"; shows DALI_Config.Szenenwert[16]; tooltip 0 % = Off 1 - 100 % = Dim level 101 % = Mask; editable
rectangle at (645,255)-(671,281): text "24"; alarm colour if Dali_Config.Kurzadr[24]
rectangle at (670,255)-(711,281): text "%s"; shows DALI_Config.Szenenwert[24]; tooltip 0 % = Off 1 - 100 % = Dim level 101 % = Mask; editable
rectangle at (645,295)-(671,321): text "32"; alarm colour if Dali_Config.Kurzadr[32]
rectangle at (670,295)-(711,321): text "%s"; shows DALI_Config.Szenenwert[32]; tooltip 0 % = Off 1 - 100 % = Dim level 101 % = Mask; editable
rectangle at (645,335)-(671,361): text "40"; alarm colour if Dali_Config.Kurzadr[40]
rectangle at (670,335)-(711,361): text "%s"; shows DALI_Config.Szenenwert[40]; tooltip 0 % = Off 1 - 100 % = Dim level 101 % = Mask; editable
rectangle at (645,375)-(671,401): text "48"; alarm colour if Dali_Config.Kurzadr[48]
rectangle at (670,375)-(711,401): text "%s"; shows DALI_Config.Szenenwert[48]; tooltip 0 % = Off 1 - 100 % = Dim level 101 % = Mask; editable
rectangle at (645,415)-(671,441): text "56"; alarm colour if Dali_Config.Kurzadr[56]
rectangle at (670,415)-(711,441): text "%s"; shows DALI_Config.Szenenwert[56]; tooltip 0 % = Off 1 - 100 % = Dim level 101 % = Mask; editable
rectangle at (645,455)-(671,481): text "64"; alarm colour if Dali_Config.Kurzadr[64]
rectangle at (670,455)-(711,481): text "%s"; shows DALI_Config.Szenenwert[64]; tooltip 0 % = Off 1 - 100 % = Dim level 101 % = Mask; editable
rectangle at (165,115)-(281,151): text "Scene:"
rectangle at (285,115)-(321,151): text "%s"; shows DALI_Config.Szene; tooltip Select scene 1 - 16; editable
rectangle at (110,505)-(261,526): text "Short address available"
rectangle at (105,535)-(291,556): text "Short address not assigned"
rectangle at (51,111)-(742,498): text "Please wait!"; invisible if NOT DALI_Config.Unsichtbar
4 more shapes without text or variables
*)

(* Visualisation Sort_short_address
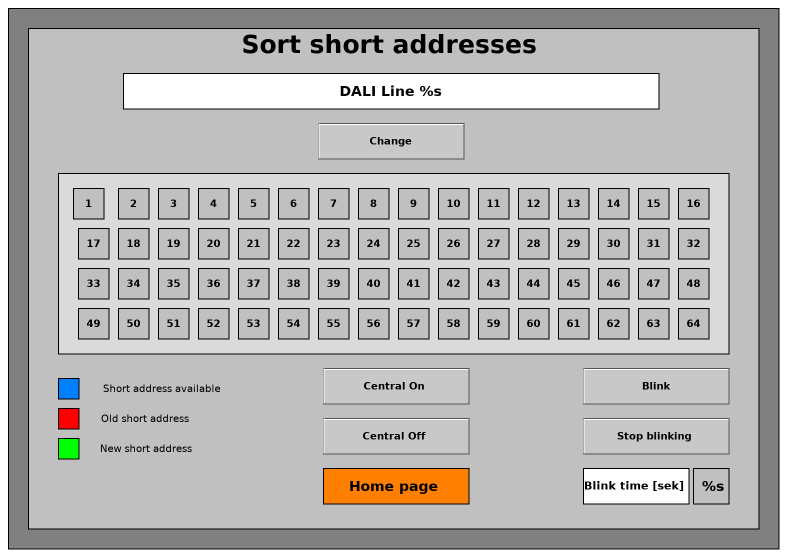
rectangle at (35,30)-(766,531): text "Sort short addresses"
rectangle at (80,190)-(111,221): text "1"; invisible if not DALI_Config.Kurzadr[1]; alarm colour if DALI_Config.mAlteAdresse[1]; toggles DALI_Config.AlteAdresse[1]
rectangle at (125,190)-(156,221): text "2"; invisible if not DALI_Config.Kurzadr[2]; alarm colour if DALI_Config.mAlteAdresse[2]; toggles DALI_Config.AlteAdresse[2]
rectangle at (165,190)-(196,221): text "3"; invisible if not DALI_Config.Kurzadr[3]; alarm colour if DALI_Config.mAlteAdresse[3]; toggles DALI_Config.AlteAdresse[3]
rectangle at (205,190)-(236,221): text "4"; invisible if not DALI_Config.Kurzadr[4]; alarm colour if DALI_Config.mAlteAdresse[4]; toggles DALI_Config.AlteAdresse[4]
rectangle at (245,190)-(276,221): text "5"; invisible if not DALI_Config.Kurzadr[5]; alarm colour if DALI_Config.mAlteAdresse[5]; toggles DALI_Config.AlteAdresse[5]
rectangle at (285,190)-(316,221): text "6"; invisible if not DALI_Config.Kurzadr[6]; alarm colour if DALI_Config.mAlteAdresse[6]; toggles DALI_Config.AlteAdresse[6]
rectangle at (325,190)-(356,221): text "7"; invisible if not DALI_Config.Kurzadr[7]; alarm colour if DALI_Config.mAlteAdresse[7]; toggles DALI_Config.AlteAdresse[7]
rectangle at (365,190)-(396,221): text "8"; invisible if not DALI_Config.Kurzadr[8]; alarm colour if DALI_Config.mAlteAdresse[8]; toggles DALI_Config.AlteAdresse[8]
rectangle at (405,190)-(436,221): text "9"; invisible if not DALI_Config.Kurzadr[9]; alarm colour if DALI_Config.mAlteAdresse[9]; toggles DALI_Config.AlteAdresse[9]
rectangle at (445,190)-(476,221): text "10"; invisible if not DALI_Config.Kurzadr[10]; alarm colour if DALI_Config.mAlteAdresse[10]; toggles DALI_Config.AlteAdresse[10]
rectangle at (485,190)-(516,221): text "11"; invisible if not DALI_Config.Kurzadr[11]; alarm colour if DALI_Config.mAlteAdresse[11]; toggles DALI_Config.AlteAdresse[11]
rectangle at (525,190)-(556,221): text "12"; invisible if not DALI_Config.Kurzadr[12]; alarm colour if DALI_Config.mAlteAdresse[12]; toggles DALI_Config.AlteAdresse[12]
rectangle at (565,190)-(596,221): text "13"; invisible if not DALI_Config.Kurzadr[13]; alarm colour if DALI_Config.mAlteAdresse[13]; toggles DALI_Config.AlteAdresse[13]
rectangle at (605,190)-(636,221): text "14"; invisible if not DALI_Config.Kurzadr[14]; alarm colour if DALI_Config.mAlteAdresse[14]; toggles DALI_Config.AlteAdresse[14]
rectangle at (645,190)-(676,221): text "15"; invisible if not DALI_Config.Kurzadr[15]; alarm colour if DALI_Config.mAlteAdresse[15]; toggles DALI_Config.AlteAdresse[15]
rectangle at (685,190)-(716,221): text "16"; invisible if not DALI_Config.Kurzadr[16]; alarm colour if DALI_Config.mAlteAdresse[16]; toggles DALI_Config.AlteAdresse[16]
rectangle at (85,230)-(116,261): text "17"; invisible if not DALI_Config.Kurzadr[17]; alarm colour if DALI_Config.mAlteAdresse[17]; toggles DALI_Config.AlteAdresse[17]
rectangle at (165,230)-(196,261): text "19"; invisible if not DALI_Config.Kurzadr[19]; alarm colour if DALI_Config.mAlteAdresse[19]; toggles DALI_Config.AlteAdresse[19]
rectangle at (125,230)-(156,261): text "18"; invisible if not DALI_Config.Kurzadr[18]; alarm colour if DALI_Config.mAlteAdresse[18]; toggles DALI_Config.AlteAdresse[18]
rectangle at (205,230)-(236,261): text "20"; invisible if not DALI_Config.Kurzadr[20]; alarm colour if DALI_Config.mAlteAdresse[20]; toggles DALI_Config.AlteAdresse[20]
rectangle at (245,230)-(276,261): text "21"; invisible if not DALI_Config.Kurzadr[21]; alarm colour if DALI_Config.mAlteAdresse[21]; toggles DALI_Config.AlteAdresse[21]
rectangle at (285,230)-(316,261): text "22"; invisible if not DALI_Config.Kurzadr[22]; alarm colour if DALI_Config.mAlteAdresse[22]; toggles DALI_Config.AlteAdresse[22]
rectangle at (325,230)-(356,261): text "23"; invisible if not DALI_Config.Kurzadr[23]; alarm colour if DALI_Config.mAlteAdresse[23]; toggles DALI_Config.AlteAdresse[23]
rectangle at (365,230)-(396,261): text "24"; invisible if not DALI_Config.Kurzadr[24]; alarm colour if DALI_Config.mAlteAdresse[24]; toggles DALI_Config.AlteAdresse[24]
rectangle at (405,230)-(436,261): text "25"; invisible if not DALI_Config.Kurzadr[25]; alarm colour if DALI_Config.mAlteAdresse[25]; toggles DALI_Config.AlteAdresse[25]
rectangle at (565,230)-(596,261): text "29"; invisible if not DALI_Config.Kurzadr[29]; alarm colour if DALI_Config.mAlteAdresse[29]; toggles DALI_Config.AlteAdresse[29]
rectangle at (525,230)-(556,261): text "28"; invisible if not DALI_Config.Kurzadr[28]; alarm colour if DALI_Config.mAlteAdresse[28]; toggles DALI_Config.AlteAdresse[28]
rectangle at (485,230)-(516,261): text "27"; invisible if not DALI_Config.Kurzadr[27]; alarm colour if DALI_Config.mAlteAdresse[27]; toggles DALI_Config.AlteAdresse[27]
rectangle at (445,230)-(476,261): text "26"; invisible if not DALI_Config.Kurzadr[26]; alarm colour if DALI_Config.mAlteAdresse[26]; toggles DALI_Config.AlteAdresse[26]
rectangle at (605,230)-(636,261): text "30"; invisible if not DALI_Config.Kurzadr[30]; alarm colour if DALI_Config.mAlteAdresse[30]; toggles DALI_Config.AlteAdresse[30]
rectangle at (645,230)-(676,261): text "31"; invisible if not DALI_Config.Kurzadr[31]; alarm colour if DALI_Config.mAlteAdresse[31]; toggles DALI_Config.AlteAdresse[31]
rectangle at (685,230)-(716,261): text "32"; invisible if not DALI_Config.Kurzadr[32]; alarm colour if DALI_Config.mAlteAdresse[32]; toggles DALI_Config.AlteAdresse[32]
rectangle at (85,270)-(116,301): text "33"; invisible if not DALI_Config.Kurzadr[33]; alarm colour if DALI_Config.mAlteAdresse[33]; toggles DALI_Config.AlteAdresse[33]
rectangle at (125,270)-(156,301): text "34"; invisible if not DALI_Config.Kurzadr[34]; alarm colour if DALI_Config.mAlteAdresse[34]; toggles DALI_Config.AlteAdresse[34]
rectangle at (205,270)-(236,301): text "36"; invisible if not DALI_Config.Kurzadr[36]; alarm colour if DALI_Config.mAlteAdresse[36]; toggles DALI_Config.AlteAdresse[36]
rectangle at (285,270)-(316,301): text "38"; invisible if not DALI_Config.Kurzadr[38]; alarm colour if DALI_Config.mAlteAdresse[38]; toggles DALI_Config.AlteAdresse[38]
rectangle at (325,270)-(356,301): text "39"; invisible if not DALI_Config.Kurzadr[39]; alarm colour if DALI_Config.mAlteAdresse[39]; toggles DALI_Config.AlteAdresse[39]
rectangle at (245,270)-(276,301): text "37"; invisible if not DALI_Config.Kurzadr[37]; alarm colour if DALI_Config.mAlteAdresse[37]; toggles DALI_Config.AlteAdresse[37]
rectangle at (165,270)-(196,301): text "35"; invisible if not DALI_Config.Kurzadr[35]; alarm colour if DALI_Config.mAlteAdresse[35]; toggles DALI_Config.AlteAdresse[35]
rectangle at (405,270)-(436,301): text "41"; invisible if not DALI_Config.Kurzadr[41]; alarm colour if DALI_Config.mAlteAdresse[41]; toggles DALI_Config.AlteAdresse[41]
rectangle at (445,270)-(476,301): text "42"; invisible if not DALI_Config.Kurzadr[42]; alarm colour if DALI_Config.mAlteAdresse[42]; toggles DALI_Config.AlteAdresse[42]
rectangle at (365,270)-(396,301): text "40"; invisible if not DALI_Config.Kurzadr[40]; alarm colour if DALI_Config.mAlteAdresse[40]; toggles DALI_Config.AlteAdresse[40]
rectangle at (485,270)-(516,301): text "43"; invisible if not DALI_Config.Kurzadr[43]; alarm colour if DALI_Config.mAlteAdresse[43]; toggles DALI_Config.AlteAdresse[43]
rectangle at (525,270)-(556,301): text "44"; invisible if not DALI_Config.Kurzadr[44]; alarm colour if DALI_Config.mAlteAdresse[44]; toggles DALI_Config.AlteAdresse[44]
rectangle at (565,270)-(596,301): text "45"; invisible if not DALI_Config.Kurzadr[45]; alarm colour if DALI_Config.mAlteAdresse[45]; toggles DALI_Config.AlteAdresse[45]
rectangle at (605,270)-(636,301): text "46"; invisible if not DALI_Config.Kurzadr[46]; alarm colour if DALI_Config.mAlteAdresse[46]; toggles DALI_Config.AlteAdresse[46]
rectangle at (645,270)-(676,301): text "47"; invisible if not DALI_Config.Kurzadr[47]; alarm colour if DALI_Config.mAlteAdresse[47]; toggles DALI_Config.AlteAdresse[47]
rectangle at (685,270)-(716,301): text "48"; invisible if not DALI_Config.Kurzadr[48]; alarm colour if DALI_Config.mAlteAdresse[48]; toggles DALI_Config.AlteAdresse[48]
rectangle at (85,310)-(116,341): text "49"; invisible if not DALI_Config.Kurzadr[49]; alarm colour if DALI_Config.mAlteAdresse[49]; toggles DALI_Config.AlteAdresse[49]
rectangle at (125,310)-(156,341): text "50"; invisible if not DALI_Config.Kurzadr[50]; alarm colour if DALI_Config.mAlteAdresse[50]; toggles DALI_Config.AlteAdresse[50]
rectangle at (165,310)-(196,341): text "51"; invisible if not DALI_Config.Kurzadr[51]; alarm colour if DALI_Config.mAlteAdresse[51]; toggles DALI_Config.AlteAdresse[51]
rectangle at (205,310)-(236,341): text "52"; invisible if not DALI_Config.Kurzadr[52]; alarm colour if DALI_Config.mAlteAdresse[52]; toggles DALI_Config.AlteAdresse[52]
rectangle at (245,310)-(276,341): text "53"; invisible if not DALI_Config.Kurzadr[53]; alarm colour if DALI_Config.mAlteAdresse[53]; toggles DALI_Config.AlteAdresse[53]
rectangle at (285,310)-(316,341): text "54"; invisible if not DALI_Config.Kurzadr[54]; alarm colour if DALI_Config.mAlteAdresse[54]; toggles DALI_Config.AlteAdresse[54]
rectangle at (325,310)-(356,341): text "55"; invisible if not DALI_Config.Kurzadr[55]; alarm colour if DALI_Config.mAlteAdresse[55]; toggles DALI_Config.AlteAdresse[55]
rectangle at (365,310)-(396,341): text "56"; invisible if not DALI_Config.Kurzadr[56]; alarm colour if DALI_Config.mAlteAdresse[56]; toggles DALI_Config.AlteAdresse[56]
rectangle at (405,310)-(436,341): text "57"; invisible if not DALI_Config.Kurzadr[57]; alarm colour if DALI_Config.mAlteAdresse[57]; toggles DALI_Config.AlteAdresse[57]
rectangle at (485,310)-(516,341): text "59"; invisible if not DALI_Config.Kurzadr[59]; alarm colour if DALI_Config.mAlteAdresse[59]; toggles DALI_Config.AlteAdresse[59]
rectangle at (525,310)-(556,341): text "60"; invisible if not DALI_Config.Kurzadr[60]; alarm colour if DALI_Config.mAlteAdresse[60]; toggles DALI_Config.AlteAdresse[60]
rectangle at (565,310)-(596,341): text "61"; invisible if not DALI_Config.Kurzadr[61]; alarm colour if DALI_Config.mAlteAdresse[61]; toggles DALI_Config.AlteAdresse[61]
rectangle at (605,310)-(636,341): text "62"; invisible if not DALI_Config.Kurzadr[62]; alarm colour if DALI_Config.mAlteAdresse[62]; toggles DALI_Config.AlteAdresse[62]
rectangle at (445,310)-(476,341): text "58"; invisible if not DALI_Config.Kurzadr[58]; alarm colour if DALI_Config.mAlteAdresse[58]; toggles DALI_Config.AlteAdresse[58]
rectangle at (645,310)-(676,341): text "63"; invisible if not DALI_Config.Kurzadr[63]; alarm colour if DALI_Config.mAlteAdresse[63]; toggles DALI_Config.AlteAdresse[63]
rectangle at (685,310)-(716,341): text "64"; invisible if not DALI_Config.Kurzadr[64]; alarm colour if DALI_Config.mAlteAdresse[64]; toggles DALI_Config.AlteAdresse[64]
rectangle at (80,190)-(111,221): text "1"; invisible if DALI_Config.Kurzadr[1]; alarm colour if DALI_Config.mNeueAdresse[1]; toggles DALI_Config.NeueAdresse[1]
rectangle at (125,190)-(156,221): text "2"; invisible if DALI_Config.Kurzadr[2]; alarm colour if DALI_Config.mNeueAdresse[2]; toggles DALI_Config.NeueAdresse[2]
rectangle at (405,190)-(436,221): text "9"; invisible if DALI_Config.Kurzadr[9]; alarm colour if DALI_Config.mNeueAdresse[9]; toggles DALI_Config.NeueAdresse[9]
rectangle at (165,190)-(196,221): text "3"; invisible if DALI_Config.Kurzadr[3]; alarm colour if DALI_Config.mNeueAdresse[3]; toggles DALI_Config.NeueAdresse[3]
rectangle at (205,190)-(236,221): text "4"; invisible if DALI_Config.Kurzadr[4]; alarm colour if DALI_Config.mNeueAdresse[4]; toggles DALI_Config.NeueAdresse[4]
rectangle at (245,190)-(276,221): text "5"; invisible if DALI_Config.Kurzadr[5]; alarm colour if DALI_Config.mNeueAdresse[5]; toggles DALI_Config.NeueAdresse[5]
rectangle at (285,190)-(316,221): text "6"; invisible if DALI_Config.Kurzadr[6]; alarm colour if DALI_Config.mNeueAdresse[6]; toggles DALI_Config.NeueAdresse[6]
rectangle at (325,190)-(356,221): text "7"; invisible if DALI_Config.Kurzadr[7]; alarm colour if DALI_Config.mNeueAdresse[7]; toggles DALI_Config.NeueAdresse[7]
rectangle at (365,190)-(396,221): text "8"; invisible if DALI_Config.Kurzadr[8]; alarm colour if DALI_Config.mNeueAdresse[8]; toggles DALI_Config.NeueAdresse[8]
rectangle at (445,190)-(476,221): text "10"; invisible if DALI_Config.Kurzadr[10]; alarm colour if DALI_Config.mNeueAdresse[10]; toggles DALI_Config.NeueAdresse[10]
rectangle at (485,190)-(516,221): text "11"; invisible if DALI_Config.Kurzadr[11]; alarm colour if DALI_Config.mNeueAdresse[11]; toggles DALI_Config.NeueAdresse[11]
rectangle at (525,190)-(556,221): text "12"; invisible if DALI_Config.Kurzadr[12]; alarm colour if DALI_Config.mNeueAdresse[12]; toggles DALI_Config.NeueAdresse[12]
rectangle at (565,190)-(596,221): text "13"; invisible if DALI_Config.Kurzadr[13]; alarm colour if DALI_Config.mNeueAdresse[13]; toggles DALI_Config.NeueAdresse[13]
rectangle at (605,190)-(636,221): text "14"; invisible if DALI_Config.Kurzadr[14]; alarm colour if DALI_Config.mNeueAdresse[14]; toggles DALI_Config.NeueAdresse[14]
rectangle at (645,190)-(676,221): text "15"; invisible if DALI_Config.Kurzadr[15]; alarm colour if DALI_Config.mNeueAdresse[15]; toggles DALI_Config.NeueAdresse[15]
rectangle at (85,230)-(116,261): text "17"; invisible if DALI_Config.Kurzadr[17]; alarm colour if DALI_Config.mNeueAdresse[17]; toggles DALI_Config.NeueAdresse[17]
rectangle at (125,230)-(156,261): text "18"; invisible if DALI_Config.Kurzadr[18]; alarm colour if DALI_Config.mNeueAdresse[18]; toggles DALI_Config.NeueAdresse[18]
rectangle at (685,190)-(716,221): text "16"; invisible if DALI_Config.Kurzadr[16]; alarm colour if DALI_Config.mNeueAdresse[16]; toggles DALI_Config.NeueAdresse[16]
rectangle at (405,230)-(436,261): text "25"; invisible if DALI_Config.Kurzadr[25]; alarm colour if DALI_Config.mNeueAdresse[25]; toggles DALI_Config.NeueAdresse[25]
rectangle at (165,230)-(196,261): text "19"; invisible if DALI_Config.Kurzadr[19]; alarm colour if DALI_Config.mNeueAdresse[19]; toggles DALI_Config.NeueAdresse[19]
rectangle at (205,230)-(236,261): text "20"; invisible if DALI_Config.Kurzadr[20]; alarm colour if DALI_Config.mNeueAdresse[20]; toggles DALI_Config.NeueAdresse[20]
rectangle at (285,230)-(316,261): text "22"; invisible if DALI_Config.Kurzadr[22]; alarm colour if DALI_Config.mNeueAdresse[22]; toggles DALI_Config.NeueAdresse[22]
rectangle at (325,230)-(356,261): text "23"; invisible if DALI_Config.Kurzadr[23]; alarm colour if DALI_Config.mNeueAdresse[23]; toggles DALI_Config.NeueAdresse[23]
rectangle at (245,230)-(276,261): text "21"; invisible if DALI_Config.Kurzadr[21]; alarm colour if DALI_Config.mNeueAdresse[21]; toggles DALI_Config.NeueAdresse[21]
rectangle at (365,230)-(396,261): text "24"; invisible if DALI_Config.Kurzadr[24]; alarm colour if DALI_Config.mNeueAdresse[24]; toggles DALI_Config.NeueAdresse[24]
rectangle at (445,230)-(476,261): text "26"; invisible if DALI_Config.Kurzadr[26]; alarm colour if DALI_Config.mNeueAdresse[26]; toggles DALI_Config.NeueAdresse[26]
rectangle at (485,230)-(516,261): text "27"; invisible if DALI_Config.Kurzadr[27]; alarm colour if DALI_Config.mNeueAdresse[27]; toggles DALI_Config.NeueAdresse[27]
rectangle at (525,230)-(556,261): text "28"; invisible if DALI_Config.Kurzadr[28]; alarm colour if DALI_Config.mNeueAdresse[28]; toggles DALI_Config.NeueAdresse[28]
rectangle at (645,230)-(676,261): text "31"; invisible if DALI_Config.Kurzadr[31]; alarm colour if DALI_Config.mNeueAdresse[31]; toggles DALI_Config.NeueAdresse[31]
rectangle at (565,230)-(596,261): text "29"; invisible if DALI_Config.Kurzadr[29]; alarm colour if DALI_Config.mNeueAdresse[29]; toggles DALI_Config.NeueAdresse[29]
rectangle at (685,230)-(716,261): text "32"; invisible if DALI_Config.Kurzadr[32]; alarm colour if DALI_Config.mNeueAdresse[32]; toggles DALI_Config.NeueAdresse[32]
rectangle at (85,270)-(116,301): text "33"; invisible if DALI_Config.Kurzadr[33]; alarm colour if DALI_Config.mNeueAdresse[33]; toggles DALI_Config.NeueAdresse[33]
rectangle at (125,270)-(156,301): text "34"; invisible if DALI_Config.Kurzadr[34]; alarm colour if DALI_Config.mNeueAdresse[34]; toggles DALI_Config.NeueAdresse[34]
rectangle at (605,230)-(636,261): text "30"; invisible if DALI_Config.Kurzadr[30]; alarm colour if DALI_Config.mNeueAdresse[30]; toggles DALI_Config.NeueAdresse[30]
rectangle at (165,270)-(196,301): text "35"; invisible if DALI_Config.Kurzadr[35]; alarm colour if DALI_Config.mNeueAdresse[35]; toggles DALI_Config.NeueAdresse[35]
rectangle at (205,270)-(236,301): text "36"; invisible if DALI_Config.Kurzadr[36]; alarm colour if DALI_Config.mNeueAdresse[36]; toggles DALI_Config.NeueAdresse[36]
rectangle at (245,270)-(276,301): text "37"; invisible if DALI_Config.Kurzadr[37]; alarm colour if DALI_Config.mNeueAdresse[37]; toggles DALI_Config.NeueAdresse[37]
rectangle at (285,270)-(316,301): text "38"; invisible if DALI_Config.Kurzadr[38]; alarm colour if DALI_Config.mNeueAdresse[38]; toggles DALI_Config.NeueAdresse[38]
rectangle at (325,270)-(356,301): text "39"; invisible if DALI_Config.Kurzadr[39]; alarm colour if DALI_Config.mNeueAdresse[39]; toggles DALI_Config.NeueAdresse[39]
rectangle at (525,270)-(556,301): text "44"; invisible if DALI_Config.Kurzadr[44]; alarm colour if DALI_Config.mNeueAdresse[44]; toggles DALI_Config.NeueAdresse[44]
rectangle at (485,270)-(516,301): text "43"; invisible if DALI_Config.Kurzadr[43]; alarm colour if DALI_Config.mNeueAdresse[43]; toggles DALI_Config.NeueAdresse[43]
rectangle at (445,270)-(476,301): text "42"; invisible if DALI_Config.Kurzadr[42]; alarm colour if DALI_Config.mNeueAdresse[42]; toggles DALI_Config.NeueAdresse[42]
rectangle at (405,270)-(436,301): text "41"; invisible if DALI_Config.Kurzadr[41]; alarm colour if DALI_Config.mNeueAdresse[41]; toggles DALI_Config.NeueAdresse[41]
rectangle at (365,270)-(396,301): text "40"; invisible if DALI_Config.Kurzadr[40]; alarm colour if DALI_Config.mNeueAdresse[40]; toggles DALI_Config.NeueAdresse[40]
rectangle at (565,270)-(596,301): text "45"; invisible if DALI_Config.Kurzadr[45]; alarm colour if DALI_Config.mNeueAdresse[45]; toggles DALI_Config.NeueAdresse[45]
rectangle at (605,270)-(636,301): text "46"; invisible if DALI_Config.Kurzadr[46]; alarm colour if DALI_Config.mNeueAdresse[46]; toggles DALI_Config.NeueAdresse[46]
rectangle at (645,270)-(676,301): text "47"; invisible if DALI_Config.Kurzadr[47]; alarm colour if DALI_Config.mNeueAdresse[47]; toggles DALI_Config.NeueAdresse[47]
rectangle at (685,270)-(716,301): text "48"; invisible if DALI_Config.Kurzadr[48]; alarm colour if DALI_Config.mNeueAdresse[48]; toggles DALI_Config.NeueAdresse[48]
rectangle at (85,310)-(116,341): text "49"; invisible if DALI_Config.Kurzadr[49]; alarm colour if DALI_Config.mNeueAdresse[49]; toggles DALI_Config.NeueAdresse[49]
rectangle at (125,310)-(156,341): text "50"; invisible if DALI_Config.Kurzadr[50]; alarm colour if DALI_Config.mNeueAdresse[50]; toggles DALI_Config.NeueAdresse[50]
rectangle at (165,310)-(196,341): text "51"; invisible if DALI_Config.Kurzadr[51]; alarm colour if DALI_Config.mNeueAdresse[51]; toggles DALI_Config.NeueAdresse[51]
rectangle at (205,310)-(236,341): text "52"; invisible if DALI_Config.Kurzadr[52]; alarm colour if DALI_Config.mNeueAdresse[52]; toggles DALI_Config.NeueAdresse[52]
rectangle at (245,310)-(276,341): text "53"; invisible if DALI_Config.Kurzadr[53]; alarm colour if DALI_Config.mNeueAdresse[53]; toggles DALI_Config.NeueAdresse[53]
rectangle at (325,310)-(356,341): text "55"; invisible if DALI_Config.Kurzadr[55]; alarm colour if DALI_Config.mNeueAdresse[55]; toggles DALI_Config.NeueAdresse[55]
rectangle at (405,310)-(436,341): text "57"; invisible if DALI_Config.Kurzadr[57]; alarm colour if DALI_Config.mNeueAdresse[57]; toggles DALI_Config.NeueAdresse[57]
rectangle at (445,310)-(476,341): text "58"; invisible if DALI_Config.Kurzadr[58]; alarm colour if DALI_Config.mNeueAdresse[58]; toggles DALI_Config.NeueAdresse[58]
rectangle at (365,310)-(396,341): text "56"; invisible if DALI_Config.Kurzadr[56]; alarm colour if DALI_Config.mNeueAdresse[56]; toggles DALI_Config.NeueAdresse[56]
rectangle at (285,310)-(316,341): text "54"; invisible if DALI_Config.Kurzadr[54]; alarm colour if DALI_Config.mNeueAdresse[54]; toggles DALI_Config.NeueAdresse[54]
rectangle at (485,310)-(516,341): text "59"; invisible if DALI_Config.Kurzadr[59]; alarm colour if DALI_Config.mNeueAdresse[59]; toggles DALI_Config.NeueAdresse[59]
rectangle at (525,310)-(556,341): text "60"; invisible if DALI_Config.Kurzadr[60]; alarm colour if DALI_Config.mNeueAdresse[60]; toggles DALI_Config.NeueAdresse[60]
rectangle at (565,310)-(596,341): text "61"; invisible if DALI_Config.Kurzadr[61]; alarm colour if DALI_Config.mNeueAdresse[61]; toggles DALI_Config.NeueAdresse[61]
rectangle at (685,310)-(716,341): text "64"; invisible if DALI_Config.Kurzadr[64]; alarm colour if DALI_Config.mNeueAdresse[64]; toggles DALI_Config.NeueAdresse[64]
rectangle at (605,310)-(636,341): text "62"; invisible if DALI_Config.Kurzadr[62]; alarm colour if DALI_Config.mNeueAdresse[62]; toggles DALI_Config.NeueAdresse[62]
rectangle at (645,310)-(676,341): text "63"; invisible if DALI_Config.Kurzadr[63]; alarm colour if DALI_Config.mNeueAdresse[63]; toggles DALI_Config.NeueAdresse[63]
button at (325,125)-(471,161): text "Change"; taps DALI_Config.Tausch; tooltip If you click the button "Change", the old short address will be replaced by the new short address.
button at (590,370)-(736,406): text "Blink"; taps DALI_Config.xBlinken; tooltip If you click the button "Blink", the selected ECG will blink as long as defined by the "Blink Time" parameter.
button at (590,420)-(736,456): text "Stop blinking"; taps DALI_Config.xBlinken_Aus; tooltip If you click the button "Stop blinking", the blinking of the ECG will stop immediately.
rectangle at (90,380)-(251,401): text "Short address available"
rectangle at (100,410)-(231,431): text "Old short address"
rectangle at (105,440)-(236,461): text "New short address"
rounded rectangle at (330,470)-(476,506): text "Home page"; opens PLC_VISU; tooltip Back to home page
rectangle at (590,470)-(696,506): text "Blink time [sek]"
rectangle at (700,470)-(736,506): text "%s"; shows DALI_Config.bBlinkzeit; tooltip Enter blink time (3 - 255 seconds); editable
button at (330,370)-(476,406): text "Central On"; taps DALI_Config.Ein; tooltip If you click the button "Central On", all lamps in the network will be switched on.
button at (330,420)-(476,456): text "Central Off"; taps DALI_Config.Aus; tooltip If you click the button "Central Off", all lamps in the network will be switched off.
rounded rectangle at (130,75)-(666,111): text "DALI Line %s"; shows DALI_Config.bDali_Linie; tooltip You can change the DALI Line only on the home page.
5 more shapes without text or variables
*)
